ABB RobotStudio station: multimove_python.rsstn

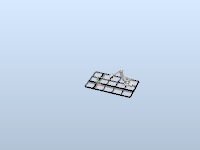
Station multimove_python (saved by RobotStudio 21.4.9700.0)
Controller MultiMove_python
  mechanical unit ROB_1: IRB1200_5_90_STD_03, 6 joints, base frame (0, 0, 0) mm
  mechanical unit ROB_2: IRB6640_180_255__04, 6 joints, base frame (3000, 1000, 0) mm, rotated rx 0 ry 0 rz 180 deg
Layout (positions relative to the parent item):
  - IRB1200_5_90_STD_03 [mechanism, from Robots\IRB1200_5_90_STD_03.rslib] at (0, 0, 0) mm; joint values [0.3678, 0.1304, 0.102, 1.0327, -0.432, -0.99] (rad or m)
  - IRB6640_180_255__04 [mechanism, from Robots\IRB6640_180_255_G_04.rslib] at (3000, 1000, 0) mm, rotated rx 0 ry 0 rz 180 deg; joint values [0.6052, 0.3981, 0.2146, -1.9801, -2.0832, 0.8515] (rad or m)
